// TIA Portal V16 export
// export: Created 2022-01-12T14:34:28.7556121Z, ExportSetting WithDefaults, DisplayName Totally Integrated Automation Portal, DisplayVersion V16 Update 4, DisplayName TIA Portal Version Control Interface, DisplayVersion V16 Update 2, DisplayName TIA Portal Openness, DisplayVersion V16 Update 4, DisplayName STEP 7 Professional, DisplayVersion V16 Update 4, DisplayName STEP 7 Safety, DisplayVersion V16, DisplayName WinCC Professional, DisplayVersion V16 Update 4
TYPE "typSygnałPomiędzyObiektamiMycia"
// stored: IsFailsafeCompliant false
   STRUCT
      toCip : "typSygnałObjectToCip";
      fromCip : "typSygnałCiToObject";
   END_STRUCT;
END_TYPE
